INTERFACE I_ExampleEquipment EXTENDS I_PackML_BaseModule

METHOD PUBLIC PickFromStagingArea : BOOL
VAR_INPUT
  orientationOfPick : ST_Orientation;
END_VAR
END_METHOD

END_INTERFACE

(* stored: Version 1.1.0.1, ProductVersion 3.1.4024.12
   Itf I_ExampleEquipment: Id {1e59db62-dd03-4efe-8704-8a3f350eee64}
   Method PickFromStagingArea: Id {0358595f-8c5b-4115-a938-7885fca2a7ea} *)
